(* CoDeSys 2.3.9.50 project: BECKHOFF.pr6 *)
(* Libraries: STANDARD.LB6 5.6.98 12:03:02 *)

(* Global variable list: TwinCAT_Import *)
VAR_GLOBAL (* DO NOT CHANGE THIS SHEET MANUALLY! *)
	PlcInVar_0	AT %QB128:	USINT;
	PlcInVar_1	AT %QB129:	USINT;
	PlcInVar_2	AT %QB130:	USINT;
	PlcInVar_3	AT %QB131:	USINT;
	PlcInVar_4	AT %QB132:	USINT;
	PlcInVar_5	AT %QB133:	USINT;
	PlcInVar_6	AT %QB134:	USINT;
	PlcInVar_7	AT %QB135:	USINT;
	PlcInVar_8	AT %QB136:	USINT;
	PlcInVar_9	AT %QB137:	USINT;
	PlcInVar_10	AT %QB138:	USINT;
	PlcInVar_11	AT %QB139:	USINT;
	PlcInVar_12	AT %QB140:	USINT;
	PlcInVar_13	AT %QB141:	USINT;
	PlcInVar_14	AT %QB142:	USINT;
	PlcInVar_15	AT %QB143:	USINT;
	PlcOutVar_0	AT %IB128:	USINT;
	PlcOutVar_1	AT %IB129:	USINT;
	PlcOutVar_2	AT %IB130:	USINT;
	PlcOutVar_3	AT %IB131:	USINT;
	PlcOutVar_4	AT %IB132:	USINT;
	PlcOutVar_5	AT %IB133:	USINT;
	PlcOutVar_6	AT %IB134:	USINT;
	PlcOutVar_7	AT %IB135:	USINT;
	PlcOutVar_8	AT %IB136:	USINT;
	PlcOutVar_9	AT %IB137:	USINT;
	PlcOutVar_10	AT %IB138:	USINT;
	PlcOutVar_11	AT %IB139:	USINT;
	PlcOutVar_12	AT %IB140:	USINT;
	PlcOutVar_13	AT %IB141:	USINT;
	PlcOutVar_14	AT %IB142:	USINT;
	PlcOutVar_15	AT %IB143:	USINT;

	Terminal_2_KL1408_1_Input_01 AT %IX0.0: BOOL; (* Water Defense *)
Terminal_2_KL1408_1_Input_02 AT %IX0.1: BOOL; (* Recovery Tank Low Level *)
Terminal_2_KL1408_1_Input_03 AT %IX0.2: BOOL; (* Recovery Tank High Level *)
Terminal_2_KL1408_1_Input_04 AT %IX0.3: BOOL; (* Recovery Tank High/High Level *)
Terminal_2_KL1408_1_Input_05 AT %IX0.4: BOOL; (* Static Reel A *)
Terminal_2_KL1408_1_Input_06 AT %IX0.5: BOOL; (* Hydrant Coupler *)
Terminal_2_KL1408_1_Input_07 AT %IX0.6: BOOL; (* Platform Position *)
	Terminal_2_KL1408_1_Input_08 AT %IX0.7: BOOL; (* Front Stabilizer Up *)

Terminal_3_KL1408_2_Input_01 AT %IX1.0: BOOL; (* Side Stabilizer Up *)
Terminal_3_KL1408_2_Input_02 AT %IX1.1: BOOL; (* Front Stabilizer Down *)
Terminal_3_KL1408_2_Input_03 AT %IX1.2: BOOL; (* Lock Inlet Extension *)
Terminal_3_KL1408_2_Input_04 AT %IX1.3: BOOL; (* Underwing Side Nozzle *)
Terminal_3_KL1408_2_Input_05 AT %IX1.4: BOOL; (* Not Assigned *)
Terminal_3_KL1408_2_Input_06 AT %IX1.5: BOOL; (* Not Assigned *)
Terminal_3_KL1408_2_Input_07 AT %IX1.6: BOOL; (* +15 Signal *)
	Terminal_3_KL1408_2_Input_08 AT %IX1.7: BOOL; (* Platform Door Lock *)

	Terminal_4_KL1408_3_Input_01 AT %IX2.0: BOOL; (* Underwing Platform Nozzle A *)
Terminal_4_KL1408_3_Input_02 AT %IX2.1: BOOL; (* Underwing Platform Nozzle B *)
Terminal_4_KL1408_3_Input_03 AT %IX2.2: BOOL; (* Laser Platform Switch *)
Terminal_4_KL1408_3_Input_04 AT %IX2.3: BOOL; (* Panel & Visual Sampler Light Switch *)
Terminal_4_KL1408_3_Input_05 AT %IX2.4: BOOL; (* Interlock Override *)
Terminal_4_KL1408_3_Input_06 AT %IX2.5: BOOL; (* Auto Start/Stop Engine Switch *)
	Terminal_4_KL1408_3_Input_07 AT %IX2.6: BOOL; (* EFSO *)
	Terminal_4_KL1408_3_Input_08 AT %IX2.7: BOOL; (* Rewind Hose Reel Switch *)

	Terminal_5_KL1408_1_Input	AT %IX0.0:	BOOL;
	Terminal_5_KL1408_2_Input	AT %IX0.1:	BOOL;
Terminal_5_KL1408_4_Input_03 AT %IX3.2: BOOL; (* Start Bartec *)
Terminal_5_KL1408_4_Input_04 AT %IX3.3: BOOL; (* DP Stop *)
Terminal_5_KL1408_4_Input_05 AT %IX3.4: BOOL; (* AFGUARD 15 PPM *)
Terminal_5_KL1408_4_Input_06 AT %IX3.5: BOOL; (* AFGUARD 30 PPM *)
Terminal_5_KL1408_4_Input_07 AT %IX3.6: BOOL; (* Air Pressure *)
	Terminal_5_KL1408_4_Input_08 AT %IX3.7: BOOL; (* Stabilizers Up Switch *)

Terminal_6_KL1408_5_Input_01 AT %IX4.0: BOOL; (* Stabilizers Down Switch *)
Terminal_6_KL1408_5_Input_02 AT %IX4.1: BOOL; (* Deadman Override Switch *)
Terminal_6_KL1408_5_Input_03 AT %IX4.2: BOOL; (* Recovery Tank Switch *)
Terminal_6_KL1408_5_Input_04 AT %IX4.3: BOOL; (* Work Light Switch *)
Terminal_6_KL1408_5_Input_05 AT %IX4.4: BOOL; (* Ultrasonic Left Platform Sensor *)
Terminal_6_KL1408_5_Input_06 AT %IX4.5: BOOL; (* Ultrasonic Right Platform Sensor *)
Terminal_6_KL1408_5_Input_07 AT %IX4.6: BOOL; (* Platform Up Switch *)
	Terminal_6_KL1408_5_Input_08 AT %IX4.7: BOOL; (* Platform Down Switch *)

Terminal_7_KL1408_6_Input_01 AT %IX5.0: BOOL; (* Limit Platform Switch *)
Terminal_7_KL1408_6_Input_02 AT %IX5.1: BOOL; (* Deadman Handle Interlock *)
Terminal_7_KL1408_6_Input_03 AT %IX5.2: BOOL; (* Deadman Handle Active *)
Terminal_7_KL1408_6_Input_04 AT %IX5.3: BOOL; (* Deadman Light Timer *)
Terminal_7_KL1408_6_Input_05 AT %IX5.4: BOOL; (* Extra Cab Input Signal *)
Terminal_7_KL1408_6_Input_06 AT %IX5.5: BOOL; (* Not Assigned *)
Terminal_7_KL1408_6_Input_07 AT %IX5.6: BOOL; (* Handbrake Active *)
Terminal_7_KL1408_6_Input_08 AT %IX5.7: BOOL; (* PTO Active *)

	Terminal_8_KL1408_1_Input	AT %IX0.0:	BOOL;
	Terminal_8_KL1408_2_Input	AT %IX0.1:	BOOL;
	Terminal_8_KL1408_3_Input	AT %IX0.2:	BOOL;
	Terminal_8_KL1408_4_Input	AT %IX0.3:	BOOL;
	Terminal_8_KL1408_5_Input	AT %IX0.4:	BOOL;
	Terminal_8_KL1408_6_Input	AT %IX0.5:	BOOL;
	Terminal_8_KL1408_7_Input	AT %IX0.6:	BOOL;
	Terminal_8_KL1408_8_Input	AT %IX0.7:	BOOL;

	Terminal_9_KL2424_1_Input	AT %IX0.0:	BOOL;
	Terminal_9_KL2424_2_Input	AT %IX0.1:	BOOL;
	Terminal_9_KL2424_3_Input	AT %IX0.2:	BOOL;
	Terminal_9_KL2424_4_Input	AT %IX0.3:	BOOL;
	Terminal_9_KL2424_5_Input	AT %IX0.4:	BOOL;
	Terminal_9_KL2424_6_Input	AT %IX0.5:	BOOL;
	Terminal_9_KL2424_7_Input	AT %IX0.6:	BOOL;
	Terminal_9_KL2424_8_Input	AT %IX0.7:	BOOL;

	Terminal_10_KL2424_1_Input	AT %IX0.0:	BOOL;
	Terminal_10_KL2424_2_Input	AT %IX0.1:	BOOL;
	Terminal_10_KL2424_3_Input	AT %IX0.2:	BOOL;
	Terminal_10_KL2424_4_Input	AT %IX0.3:	BOOL;
	Terminal_10_KL2424_5_Input	AT %IX0.4:	BOOL;
	Terminal_10_KL2424_6_Input	AT %IX0.5:	BOOL;
	Terminal_10_KL2424_7_Input	AT %IX0.6:	BOOL;
	Terminal_10_KL2424_8_Input	AT %IX0.7:	BOOL;

	Terminal_11_KL2424_1_Input	AT %IX0.0:	BOOL;
	Terminal_11_KL2424_2_Input	AT %IX0.1:	BOOL;
	Terminal_11_KL2424_3_Input	AT %IX0.2:	BOOL;
	Terminal_11_KL2424_4_Input	AT %IX0.3:	BOOL;
	Terminal_11_KL2424_5_Input	AT %IX0.4:	BOOL;
	Terminal_11_KL2424_6_Input	AT %IX0.5:	BOOL;
	Terminal_11_KL2424_7_Input	AT %IX0.6:	BOOL;
	Terminal_11_KL2424_8_Input	AT %IX0.7:	BOOL;

	Terminal_12_KL2424_1_Input	AT %IX0.0:	BOOL;
	Terminal_12_KL2424_2_Input	AT %IX0.1:	BOOL;
	Terminal_12_KL2424_3_Input	AT %IX0.2:	BOOL;
	Terminal_12_KL2424_4_Input	AT %IX0.3:	BOOL;
	Terminal_12_KL2424_5_Input	AT %IX0.4:	BOOL;
	Terminal_12_KL2424_6_Input	AT %IX0.5:	BOOL;
	Terminal_12_KL2424_7_Input	AT %IX0.6:	BOOL;
	Terminal_12_KL2424_8_Input	AT %IX0.7:	BOOL;

	Terminal_13_KL2408_1_Output	AT %QX0.0:	BOOL;
	Terminal_13_KL2408_2_Input	AT %QX0.1:	BOOL;
	Terminal_13_KL2408_3_Input	AT %QX0.2:	BOOL;
	Terminal_13_KL2408_4_Input	AT %QX0.3:	BOOL;
	Terminal_13_KL2408_5_Input	AT %QX0.4:	BOOL;
	Terminal_13_KL2408_6_Input	AT %QX0.5:	BOOL;
	Terminal_13_KL2408_7_Input	AT %QX0.6:	BOOL;
	Terminal_13_KL2408_8_Input	AT %QX0.7:	BOOL;

	Terminal_14_KL2408_1_Input	AT %QX0.0:	BOOL;
	Terminal_14_KL2408_2_Input	AT %QX0.1:	BOOL;
	Terminal_14_KL2408_3_Input	AT %QX0.2:	BOOL;
	Terminal_14_KL2408_4_Input	AT %QX0.3:	BOOL;
	Terminal_14_KL2408_5_Input	AT %QX0.4:	BOOL;
	Terminal_14_KL2408_6_Input	AT %QX0.5:	BOOL;
	Terminal_14_KL2408_7_Input	AT %QX0.6:	BOOL;
	Terminal_14_KL2408_8_Input	AT %QX0.7:	BOOL;

	Terminal_15_KL2408_1_Input	AT %QX0.0:	BOOL;
	Terminal_15_KL2408_2_Input	AT %QX0.1:	BOOL;
	Terminal_15_KL2408_3_Input	AT %QX0.2:	BOOL;
	Terminal_15_KL2408_4_Input	AT %QX0.3:	BOOL;
	Terminal_15_KL2408_5_Input	AT %QX0.4:	BOOL;
	Terminal_15_KL2408_6_Input	AT %QX0.5:	BOOL;
	Terminal_15_KL2408_7_Input	AT %QX0.6:	BOOL;
	Terminal_15_KL2408_8_Input	AT %QX0.7:	BOOL;


	Terminal_16_KL2408_1_Input	AT %QX0.0:	BOOL;
	Terminal_16_KL2408_2_Input	AT %QX0.1:	BOOL;
	Terminal_16_KL2408_3_Input	AT %QX0.2:	BOOL;
	Terminal_16_KL2408_4_Input	AT %QX0.3:	BOOL;
	Terminal_16_KL2408_5_Input	AT %QX0.4:	BOOL;
	Terminal_16_KL2408_6_Input	AT %QX0.5:	BOOL;
	Terminal_16_KL2408_7_Input	AT %QX0.6:	BOOL;
	Terminal_16_KL2408_8_Input	AT %QX0.7:	BOOL;


	Terminal_17_KL2408_1_Input	AT %QX0.0:	BOOL;
	Terminal_17_KL2408_2_Input	AT %QX0.1:	BOOL;
	Terminal_17_KL2408_3_Input	AT %QX0.2:	BOOL;
	Terminal_17_KL2408_4_Input	AT %QX0.3:	BOOL;
	Terminal_17_KL2408_5_Input	AT %QX0.4:	BOOL;
	Terminal_17_KL2408_6_Input	AT %QX0.5:	BOOL;
	Terminal_17_KL2408_7_Input	AT %QX0.6:	BOOL;
	Terminal_17_KL2408_8_Input	AT %QX0.7:	BOOL;


	Terminal_18_KL2408_1_Input	AT %QX0.0:	BOOL;
	Terminal_18_KL2408_2_Input	AT %QX0.1:	BOOL;
	Terminal_18_KL2408_3_Input	AT %QX0.2:	BOOL;
	Terminal_18_KL2408_4_Input	AT %QX0.3:	BOOL;
	Terminal_18_KL2408_5_Input	AT %QX0.4:	BOOL;
	Terminal_18_KL2408_6_Input	AT %QX0.5:	BOOL;
	Terminal_18_KL2408_7_Input	AT %QX0.6:	BOOL;
	Terminal_18_KL2408_8_Input	AT %QX0.7:	BOOL;




 END_VAR

(* POU MAIN, LD *)
PROGRAM MAIN
VAR
END_VAR
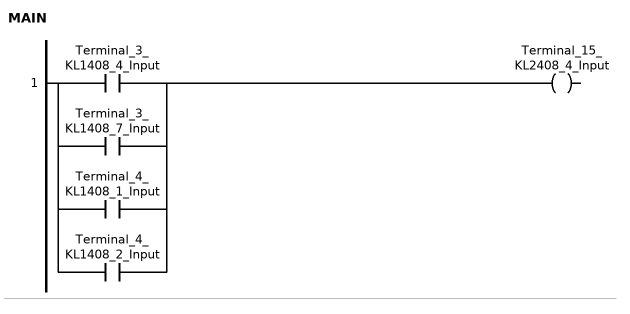
_LD_ (* Ladder Diagram *)
NETWORK 1
	{ [Terminal_3_KL1408_4_Input] | [Terminal_3_KL1408_7_Input] | [Terminal_4_KL1408_1_Input] | [Terminal_4_KL1408_2_Input] } --- (Terminal_15_KL2408_4_Input)
_END_LD_
(* the same logic as Structured Text *)
(* Network 1 *)
Terminal_15_KL2408_4_Input := Terminal_3_KL1408_4_Input OR Terminal_3_KL1408_7_Input OR Terminal_4_KL1408_1_Input OR Terminal_4_KL1408_2_Input;
END_PROGRAM
